// Mitsubishi GX Works2 project: 241111_PLC_Practice2   PLC: Q02U

PROGRAM MAIN
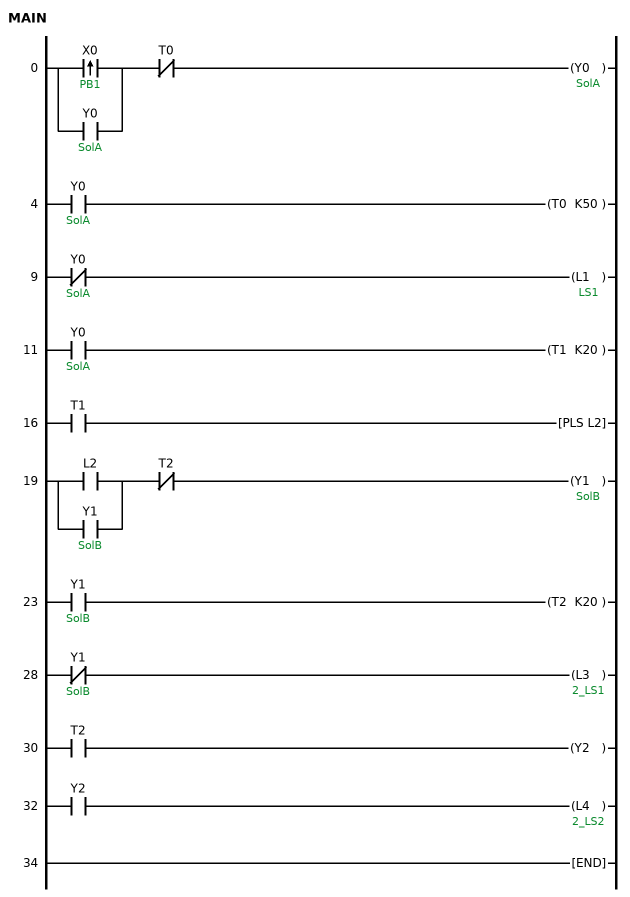
0     LDP     X0  ; PB1
      OR      Y0  ; SolA
      ANI     T0
      OUT     Y0  ; SolA
4     LD      Y0  ; SolA
      OUT     T0 K50
9     LDI     Y0  ; SolA
      OUT     L1  ; LS1
11    LD      Y0  ; SolA
      OUT     T1 K20
16    LD      T1
      PLS     L2
19    LD      L2
      OR      Y1  ; SolB
      ANI     T2
      OUT     Y1  ; SolB
23    LD      Y1  ; SolB
      OUT     T2 K20
28    LDI     Y1  ; SolB
      OUT     L3  ; 2_LS1
30    LD      T2
      OUT     Y2
32    LD      Y2
      OUT     L4  ; 2_LS2
34    END
END_PROGRAM
